// TIA Portal V17 export
// export: Created 2023-03-06T01:51:54.570799Z, ExportSetting WithDefaults, DisplayName Totally Integrated Automation Portal, DisplayVersion V17 Update 4, DisplayName TIA Portal Openness, DisplayVersion V17 Update 4, DisplayName TIA Portal Version Control Interface, DisplayVersion V17, DisplayName STEP 7 Professional, DisplayVersion V17 Update 4, DisplayName STEP 7 Safety, DisplayVersion V17, DisplayName WinCC Professional, DisplayVersion V17 Update 4
VAR_GLOBAL   // PLC tag table "Rack Variables"
   "Emergency push button PWCLH0" AT %I50.0 : Bool;   // xFDI_Slot01_In01_127S1
   "Emergency stop feedback contactors" AT %I50.1 : Bool;   // xFDI_Slot01_In03_517k1
   "Emergency stop from fire detection system" AT %I50.5 : Bool;   // xFDI_Slot01_In04_081k3
   "Push button emergency reset" AT %I50.2 : Bool;   // xFDI_Slot01_In05_513P1
   Spare AT %I50.6 : Bool;   // xFDI_Slot01_In06_Xxxxxx
   "Emergency push button PWCRH0" AT %I50.3 : Bool;   // xFDI_Slot01_In07_227S1
   "Emergency stop from PCS1 (PE)" AT %I56.0 : Bool;   // xFDI_Slot02_In01_EPCS1
   "Emergency stop from PCS2 (PE) (future expansion)" AT %I56.4 : Bool;   // xFDI_Slot02_In02_EPCS2
   "Emergency stop from External (future expansion)" AT %I56.1 : Bool;   // xFDI_Slot02_In03_EExt
   "PWCLH0 Common mode signal" AT %I56.5 : Bool;   // xFDI_Slot02_In04_125A3
   "PWCRH0 Common mode signal" AT %I56.2 : Bool;   // xFDI_Slot02_In05_225A3
   "Spare(1)" AT %I56.6 : Bool;   // xFDI_Slot02_In06_Xxxxxx
   "Spare(2)" AT %I56.3 : Bool;   // xFDI_Slot02_In07_Xxxxxx
   "Spare(3)" AT %I56.7 : Bool;   // xFDI_Slot02_In08_Xxxxxx
   "Emergency stop delayed" AT %Q62.0 : Bool;   // xFDO_Slot03_Out01_517k1
   "Emergency stop instantaneous" AT %Q62.1 : Bool;   // xFDO_Slot03_Out02_517k2
   "Emergency stop PCS1 (PE)" AT %Q62.2 : Bool;   // xFDO_Slot03_Out03_517k3
   "Emergency stop PCS1 (PE) (future expansion)" AT %Q62.3 : Bool;   // xFDO_Slot03_Out04_517k4
   "Emergency stop disconnector PWCLH0" AT %Q62.4 : Bool;   // xFDO_Slot03_Out05_517k5
   "Emergency stop disconnector PWCRH0" AT %Q62.5 : Bool;   // xFDO_Slot03_Out06_517k6
   "Emergency stop HVAC and internal fans" AT %Q62.6 : Bool;   // xFDO_Slot03_Out07_517k7
   "Light emergency reset" AT %Q62.7 : Bool;   // xFDO_Slot03_Out08_513P1
   "400 Vac Surge suppressor" AT %I0.0 : Bool;   // xDI_Slot04_In01_001F1
   "Main circuit breaker" AT %I0.1 : Bool;   // xDI_Slot04_In02_003Q1
   "Power supply Chiller CATL LH side" AT %I0.2 : Bool;   // xDI_Slot04_In03_011F1
   "Power supply Chiller CATL RH side" AT %I0.3 : Bool;   // xDI_Slot04_In04_017F1
   "Power supply HVAC PEMS" AT %I0.4 : Bool;   // xDI_Slot04_In05_023Q1
   "Power supply fans internal board" AT %I0.5 : Bool;   // xDI_Slot04_In06_025F1
   "Power supply spare" AT %I0.6 : Bool;   // xDI_Slot04_In07_025F2
   "Power supply fire detection board" AT %I0.7 : Bool;   // xDI_Slot04_In08_101F8
   "Main circuit breaker from backup diesel generator" AT %I1.0 : Bool;   // xDI_Slot05_In01_101F5
   "UPS Surge suppressor" AT %I1.1 : Bool;   // xDI_Slot05_In02_101F3
   "General breaker output UPS" AT %I1.2 : Bool;   // xDI_Slot05_In03_103F1
   "Main circuit breaker from normal power supply" AT %I1.3 : Bool;   // xDI_Slot05_In04_101F2
   "Power supply control CATL LH side" AT %I1.4 : Bool;   // xDI_Slot05_In05_105F1
   "Power supply control CATL RH side" AT %I1.5 : Bool;   // xDI_Slot05_In06_107F1
   "HVAC signal" AT %I1.6 : Bool;   // xDI_Slot05_In07_011M1
   "Power supply Unit 1 230Vac / 24Vdc" AT %I1.7 : Bool;   // xDI_Slot05_In08_109F2
   "Power supply Unit 2 230Vac / 24Vdc" AT %I2.0 : Bool;   // xDI_Slot06_In01_109F3
   "Power supply shunt opening release" AT %I2.1 : Bool;   // xDI_Slot06_In02_109F4
   "Power supply spare(1)" AT %I2.2 : Bool;   // xDI_Slot06_In03_109F5
   "Power supply 24 Vdc spare" AT %I2.3 : Bool;   // xDI_Slot06_In04_301F10
   "Power supply 24 Vdc communication equipment" AT %I2.4 : Bool;   // xDI_Slot06_In05_301F1
   "Power supply 24 Vdc safety PLC cards" AT %I2.5 : Bool;   // xDI_Slot06_In06_301F2
   "Power supply 24 Vdc digital PLC cards" AT %I2.6 : Bool;   // xDI_Slot06_In07_301F3
   "Power supply 24 Vdc common mode sensors" AT %I2.7 : Bool;   // xDI_Slot06_In08_301F4
   "Power supply 24 Vdc PLC I/O internal" AT %I3.0 : Bool;   // xDI_Slot07_In01_301F5
   "Power supply 24 Vdc PLC I/O external" AT %I3.1 : Bool;   // xDI_Slot07_In02_301F6
   "Power supply 24 Vdc fire detection system" AT %I3.2 : Bool;   // xDI_Slot07_In03_301F7
   "UPS low battery" AT %I3.3 : Bool;   // xDI_Slot07_In04_103A1
   "UPS fault" AT %I3.4 : Bool;   // xDI_Slot07_In05_103A1
   "UPS on battery" AT %I3.5 : Bool;   // xDI_Slot07_In06_103A1
   "UPS alarm" AT %I3.6 : Bool;   // xDI_Slot07_In07_103A1
   "UPS on bypass" AT %I3.7 : Bool;   // xDI_Slot07_In08_103A1
   "Power supply 24 Vdc MBMU / ETH CATL LH side" AT %I4.0 : Bool;   // xDI_Slot08_In01_301F8
   "Power supply 24 Vdc MBMU / ETH CATL RH side" AT %I4.1 : Bool;   // xDI_Slot08_In02_301F9
   "Bypass incoming line UPS from grid line" AT %I4.2 : Bool;   // xDI_Slot08_In03_101Q1
   "Bypass incoming line UPS from generator line" AT %I4.3 : Bool;   // xDI_Slot08_In04_101Q2
   "Spare(4)" AT %I4.4 : Bool;   // xDI_Slot08_In05_Xxxxx
   "Spare(5)" AT %I4.5 : Bool;   // xDI_Slot08_In06_Xxxxx
   "Spare(6)" AT %I4.6 : Bool;   // xDI_Slot08_In07_Xxxxx
   "Spare(7)" AT %I4.7 : Bool;   // xDI_Slot08_In08_Xxxxx
   "Thermostat inside PEMS threshold 40 °C" AT %I5.0 : Bool;   // xDI_Slot09_In01_531S1
   "Thermostat inside PEMS threshold 55 °C" AT %I5.1 : Bool;   // xDI_Slot09_In02_531S2
   "Panel opened PWCLH0" AT %I5.2 : Bool;   // xDI_Slot09_In03_531S3
   "Panel 1 opened PEMS" AT %I5.3 : Bool;   // xDI_Slot09_In04_531S4
   "Panel 2 opened PEMS" AT %I5.4 : Bool;   // xDI_Slot09_In05_531S5
   "Panel opened PWCRH0" AT %I5.5 : Bool;   // xDI_Slot09_In06_531S6
   "Spare(8)" AT %I5.6 : Bool;   // xDI_Slot09_In07_Xxxxx
   "Spare(9)" AT %I5.7 : Bool;   // xDI_Slot09_In08_Xxxxx
   "General fault fire detection system" AT %I6.0 : Bool;   // xDI_Slot10_In01_081k1
   "NAC alarm fire detection system" AT %I6.1 : Bool;   // xDI_Slot10_In02_081k2
   "General disconnector closed PWCLH0" AT %I6.2 : Bool;   // xDI_Slot10_In03_121Q1
   "Surge suppressor PWCLH0" AT %I6.3 : Bool;   // xDI_Slot10_In04_125F3
   "General disconnector closed PWCRH0" AT %I6.4 : Bool;   // xDI_Slot10_In05_221Q1
   "Surge suppressor PWCRH0" AT %I6.5 : Bool;   // xDI_Slot10_In06_225F3
   "Spare(10)" AT %I6.6 : Bool;   // xDI_Slot10_In07_Xxxxx
   "Spare(11)" AT %I6.7 : Bool;   // xDI_Slot10_In08_Xxxxx
   "Power supply control CATL LH side(1)" AT %Q0.0 : Bool;   // xDO_Slot11_Out01_551Q1
   "Power supply control CATL RH side(1)" AT %Q0.1 : Bool;   // xDO_Slot11_Out02_551Q2
   "Spare(12)" AT %Q0.2 : Bool;   // xDO_Slot11_Out03_551k1
   "Spare(13)" AT %Q0.3 : Bool;   // xDO_Slot11_Out04_551k2
   "UPS shut down any mode" AT %Q0.4 : Bool;   // xDO_Slot11_Out05_551k3
   "Light DC power on Battery bank LH side" AT %Q0.5 : Bool;   // xDO_Slot11_Out06_551k4
   "Light DC power on Battery bank RH side" AT %Q0.6 : Bool;   // xDO_Slot11_Out07_551k5
   "Spare(14)" AT %Q0.7 : Bool;   // xDO_Slot11_Out08_551k6
END_VAR
